{attribute 'GeneratedUsingTerminal: EL5122-0000-0016'}
{attribute addProperty BoxType "EL5122-0000-0016"}
{attribute addProperty Id "StatusAT %I*Status_770B523112Counter_valueAT %I*UDINT4Latch_valueAT %I*UDINT4"}
{attribute addProperty CRC "82931648"}
{attribute addProperty Size "20"}
TYPE ENC_Status_Channel_04F16FC0 EXTENDS InputBase_8311D824 :
STRUCT
	{attribute addProperty Name "Status"}
	Status AT %I* : Status_770B5231;
	{attribute addProperty Name "Counter_value"}
	Counter_value AT %I* : UDINT;
	{attribute addProperty Name "Latch_value"}
	Latch_value AT %I* : UDINT;
END_STRUCT
END_TYPE

(* stored: Version 1.2.0.0, ProductVersion 3.1.4024.9
   DUT ENC_Status_Channel_04F16FC0: Id {3d466e09-56eb-4dfd-a271-ce6709977571} *)
